TYPE PLCRobotOrder :
STRUCT
	GotoHome: OrderPLC;
	GotoAGVPos: OrderPLC;
	GotoBuffer: OrderPLC;
	GotoScanner: OrderPLC;
	GotoTable: OrderPLC;
END_STRUCT
END_TYPE

(* stored: Version 1.1.0.1, ProductVersion 3.1.4022.16
   DUT PLCRobotOrder: Id {8a658890-efd9-4ef4-bf0b-bdfc96b56b89} *)
